Fanuc KAREL source: hash.kl

PROGRAM hash
%NOLOCKGROUP

%INCLUDE hash.klt

%INCLUDE strings.klh
%INCLUDE hash.private.klh
%INCLUDE hash.klh

BEGIN
END hash

--Private Members

ROUTINE djb2
VAR
	hash : INTEGER
	i    : INTEGER
	char : INTEGER
BEGIN
	hash = 5381
	FOR i=1 TO STR_LEN(str) DO
		char = ORD(str, i)
		hash = hash * 33 + char
	ENDFOR
	RETURN(hash)
END djb2

-- From Java 1.5 string library
ROUTINE jsStrHash
VAR
	hash : INTEGER
	i    : INTEGER
BEGIN
	hash = 0
	FOR i=1 TO STR_LEN(str) DO
		hash = (31 * hash) + ord(str, i)
	ENDFOR
	RETURN(hash)
END jsStrHash

ROUTINE hModHash
VAR
	hash : INTEGER
BEGIN
	hash = jsStrHash(key)
	RETURN(hash MOD len + 1)
END hModHash

ROUTINE hGetIndex
VAR
	hash      : INTEGER
	tblLength : INTEGER
	index     : INTEGER
	count     : INTEGER
BEGIN
	hash = jsStrHash(key)
	tblLength = ARRAY_LEN(tbl)
	index = hash MOD tblLength + 1

	FOR count=0 TO tblLength DO
		IF UNINIT(tbl[index].key) THEN tbl[index].key = ''; ENDIF

		IF get THEN
			-- get requests require key=key
			IF ((tbl[index].key=key)) THEN
				RETURN(index)
			ENDIF
		ELSE
			-- put requests require key=key or empty
			IF ((tbl[index].key=key) OR
				(tbl[index].key='')) THEN
				RETURN(index)
			ENDIF
		ENDIF

		index = index + 1
		IF index > tblLength THEN
			index = 1
		ENDIF
	ENDFOR

	-- did not find index
	RETURN(0)
END hGetIndex


ROUTINE hPut
VAR
	index : INTEGER
BEGIN
	index = hGetIndex(key, false, tbl)
	IF index > 0 THEN
		tbl[index].key = key
		tbl[index].val = value
		RETURN(TRUE)
	ELSE
		RETURN(FALSE)
	ENDIF
END hPut

ROUTINE hGet
VAR
	index : INTEGER
BEGIN
	index = hGetIndex(key, true, tbl)
	IF index > 0 THEN
		RETURN(tbl[index].val)
	ENDIF

	RETURN('')
END hGet

ROUTINE hDel
VAR
	index : INTEGER
BEGIN
	index = hGetIndex(key, true, tbl)
	IF index > 0 THEN
		IF ((tbl[index].key=key)) THEN
			tbl[index].key = ''
      tbl[index].val = ''
			RETURN(TRUE)
		ENDIF
	ENDIF

	RETURN(FALSE)
END hDel

--Public Members

ROUTINE hashPut
VAR
	entry : INTEGER
BEGIN
	IF (key='') THEN RETURN(FALSE); ENDIF

	RETURN(hPut(key, value, BYNAME(tblProg, tblName, entry)))
END hashPut


ROUTINE hashGet
VAR
	entry : INTEGER
BEGIN
	IF (key='') THEN RETURN(''); ENDIF

	RETURN (hGet(key, BYNAME(tblProg, tblName, entry)))
END hashGet

ROUTINE hashDel
VAR
	entry : INTEGER
BEGIN
	IF (key='') THEN RETURN(FALSE); ENDIF

	RETURN (hDel(key, BYNAME(tblProg, tblName, entry)))
END hashDel
